// TIA Portal V19 export
TYPE "LEXCHANGETRAY_typeSr1000ProfinetTelegram_completionClearControlBits"
// stored: Access Published
   STRUCT
      controlByte : Byte;
      readCompleteClear : Bool;
      presetCompleteClear : Bool;
      registerPresetDataCmpltClr : Bool;
      tuneCmpltClr : Bool;
      extReqCmpltClr : Bool;
   END_STRUCT;
END_TYPE
